FUNCTION_BLOCK POST_AGGREGATOR
  {SET_ATTRIBUTE(OpcUa, SERVICE)}
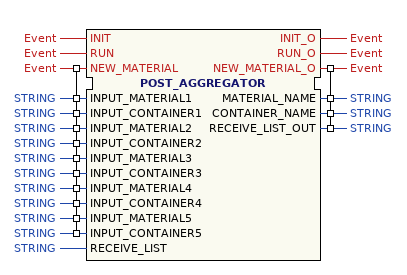
  EVENT_INPUT
    INIT;
    RUN; {SET_ATTRIBUTE(OpcUa, Method)}
    NEW_MATERIAL WITH INPUT_MATERIAL1, INPUT_CONTAINER1, INPUT_MATERIAL2, INPUT_CONTAINER2, INPUT_MATERIAL3, INPUT_CONTAINER3, INPUT_MATERIAL4, INPUT_CONTAINER4, INPUT_MATERIAL5, INPUT_CONTAINER5;
  END_EVENT
  EVENT_OUTPUT
    INIT_O;
    RUN_O;
    NEW_MATERIAL_O WITH MATERIAL_NAME, CONTAINER_NAME, RECEIVE_LIST_OUT;
  END_EVENT
  VAR_INPUT
    INPUT_MATERIAL1 : STRING; {SET_ATTRIBUTE(OpcUa, Variable.RUN)}
    INPUT_CONTAINER1 : STRING; {SET_ATTRIBUTE(OpcUa, Variable.RUN)}
    INPUT_MATERIAL2 : STRING; {SET_ATTRIBUTE(OpcUa, Variable.RUN)}
    INPUT_CONTAINER2 : STRING; {SET_ATTRIBUTE(OpcUa, Variable.RUN)}
    INPUT_MATERIAL3 : STRING; {SET_ATTRIBUTE(OpcUa, Variable.RUN)}
    INPUT_CONTAINER3 : STRING; {SET_ATTRIBUTE(OpcUa, Variable.RUN)}
    INPUT_MATERIAL4 : STRING; {SET_ATTRIBUTE(OpcUa, Variable.RUN)}
    INPUT_CONTAINER4 : STRING; {SET_ATTRIBUTE(OpcUa, Variable.RUN)}
    INPUT_MATERIAL5 : STRING; {SET_ATTRIBUTE(OpcUa, Variable.RUN)}
    INPUT_CONTAINER5 : STRING; {SET_ATTRIBUTE(OpcUa, Variable.RUN)}
    RECEIVE_LIST : STRING; {SET_ATTRIBUTE(OpcUa, Constant.RUN)}
  END_VAR
  VAR_OUTPUT
    MATERIAL_NAME : STRING; {SET_ATTRIBUTE(OpcUa, Variable.RUN)}
    CONTAINER_NAME : STRING; {SET_ATTRIBUTE(OpcUa, Variable.RUN)}
    RECEIVE_LIST_OUT : STRING; {SET_ATTRIBUTE(OpcUa, Constant.RUN)}
  END_VAR
END_FUNCTION_BLOCK
